// TIA Portal project "pick and place 3" (V16)

(* hardware
DEVICE "S7-1200-Station_1"  S7-1200 Station
   slot 0: "Baugruppenträger_0"  S7-1200 Rack  Rack  V1.0
   slot 1: "PLC_1"  CPU 1211C DC/DC/DC  6ES7 211-1AE40-0XB0  V4.1
*)

// ===== PLC "PLC_1"  CPU 1211C DC/DC/DC =====

VAR_GLOBAL   // PLC tag table "Default tag table"
   ""start"" AT %I0.0 : Bool;
   ""z sensor"" AT %I0.1 : Bool;
   ""diffuse sens"" AT %I0.2 : Bool;
   ""box detecd"" AT %I0.3 : Bool;
   ""x sensor"" AT %I0.4 : Bool;
   ""diffues2"" AT %I0.5 : Bool;
   ""stop"" AT %I0.6 : Bool;
   ""conv"" AT %Q0.0 : Bool;
   ""emitter"" AT %Q0.1 : Bool;
   ""z down"" AT %Q0.2 : Bool;
   ""grab"" AT %Q0.3 : Bool;
   ""x move"" AT %Q0.4 : Bool;
   ""conv2"" AT %Q0.5 : Bool;
   ""emitter2"" AT %Q0.6 : Bool;
END_VAR